{attribute 'GeneratedUsingTerminal: AX8118-0100-0102-0102'}
{attribute addProperty BoxType "AX8118-0100-0102-0102"}
{attribute addProperty Description "AX8118-0100-0102"}
{attribute addProperty Physics "KK"}
{attribute addProperty Id "DeviceDevice_6E2575772Device_SafetyDevice_Safety_C21945A160Ch_ACh_A_D18C6F1622WcStateAT %I*WcState_B516A2644InfoDataAT %I*InfoData_358A59CF25"}
{attribute addProperty CRC "4154992789"}
{attribute addProperty Size "113"}
TYPE AX8118_F7A82895 EXTENDS EtcSlaveTerminalBase_947E5A46 :
STRUCT
	{attribute addProperty Name "Device"}
	Device : Device_6E257577;
	{attribute addProperty Name "Device_Safety"}
	Device_Safety : Device_Safety_C21945A1;
	{attribute addProperty Name "Ch_A"}
	Ch_A : Ch_A_D18C6F16;
	{attribute addProperty Name "WcState"}
	WcState : WcState_B516A264;
	{attribute addProperty Name "InfoData"}
	InfoData : InfoData_358A59CF;
END_STRUCT
END_TYPE

(* stored: Version 1.2.0.0, ProductVersion 3.1.4024.11
   DUT AX8118_F7A82895: Id {d0ca64f4-e58f-4e2c-b99e-9e4976d7fecc} *)
